ABB RobotStudio station: DeskDome.rspag

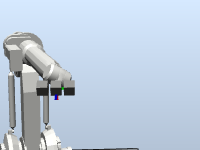
--- station ---
Station DeskDome (saved by RobotStudio 6.8.8148.134)
Controller DeskSystem
  mechanical unit ROB_1: IRB1410_5_144__01, 6 joints, base frame (0, 0, 0) mm
Layout (positions relative to the parent item):
  - IRB1410_5_144__01 [mechanism, from Robots\IRB1410_5_144_G_01.rslib] at (0, 0, 0) mm; joint values [0.3206, 0.0673, 0.0661, -0.5505, 0.5489, 0.6469] (rad or m)
  - 气缸3 [part] at (956.26, 325.16, 1145.27) mm, rotated rx -180 ry 60 rz 180 deg
  - 气缸2 [part] at (956.32, 263.96, 1145.39) mm, rotated rx -180 ry 60 rz 180 deg
  - 气缸1 [part] at (956.53, 200.68, 1145.75) mm, rotated rx -180 ry 60 rz 180 deg
  - 气缸运动 [smart component]
      signals: DI di_1, DI di_2, DI di_3, DO do_1, DO do_2, DO do_3, DI di_reset, DI di_M1, DI di_M2, DI di_M3, DO do_M1, DO do_M2, DO do_M3
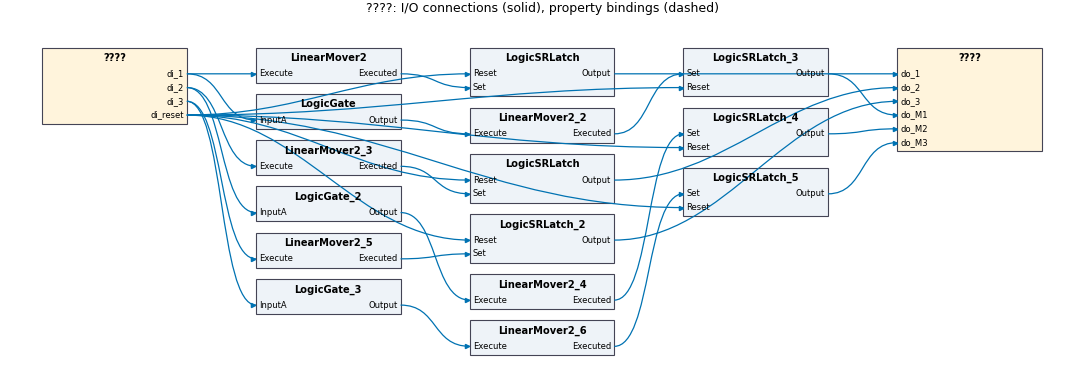
      connections:
        气缸运动.di_1 -> LinearMover2.Execute
        气缸运动.di_2 -> LinearMover2_3.Execute
        气缸运动.di_3 -> LinearMover2_5.Execute
        LogicSRLatch.Output -> 气缸运动.do_1
        气缸运动.di_reset -> LogicSRLatch.Reset
        LogicSRLatch.Output -> 气缸运动.do_2
        LogicSRLatch_2.Output -> 气缸运动.do_3
        气缸运动.di_reset -> LogicSRLatch.Reset
        气缸运动.di_reset -> LogicSRLatch_2.Reset
        LinearMover2.Executed -> LogicSRLatch.Set
        LinearMover2_2.Executed -> LogicSRLatch_3.Set
        气缸运动.di_reset -> LogicSRLatch_3.Reset
        LogicSRLatch_3.Output -> 气缸运动.do_M1
        LinearMover2_3.Executed -> LogicSRLatch.Set
        LinearMover2_4.Executed -> LogicSRLatch_4.Set
        气缸运动.di_reset -> LogicSRLatch_4.Reset
        LogicSRLatch_4.Output -> 气缸运动.do_M2
        LinearMover2_5.Executed -> LogicSRLatch_2.Set
        LinearMover2_6.Executed -> LogicSRLatch_5.Set
        气缸运动.di_reset -> LogicSRLatch_5.Reset
        LogicSRLatch_5.Output -> 气缸运动.do_M3
        气缸运动.di_1 -> LogicGate.InputA
        LogicGate.Output -> LinearMover2_2.Execute
        气缸运动.di_2 -> LogicGate_2.InputA
        LogicGate_2.Output -> LinearMover2_4.Execute
        气缸运动.di_3 -> LogicGate_3.InputA
        LogicGate_3.Output -> LinearMover2_6.Execute
    - LinearMover2 [smart component, from Components\LinearMover2.rslib]
        properties: Object=气缸1; Direction=[0 0 -0.01]; Distance=0.02; Duration=1; Reference=Global; ReferenceObject=(none)
    - LinearMover2_2 [smart component, from Components\LinearMover2.rslib]
        properties: Object=气缸1; Direction=[0 0 0.01]; Distance=0.02; Duration=1; Reference=Global; ReferenceObject=(none)
    - LinearMover2_3 [smart component, from Components\LinearMover2.rslib]
        properties: Object=气缸2; Direction=[0 0 -0.01]; Distance=0.02; Duration=1; Reference=Global; ReferenceObject=(none)
    - LinearMover2_4 [smart component, from Components\LinearMover2.rslib]
        properties: Object=气缸2; Direction=[0 0 0.01]; Distance=0.02; Duration=1; Reference=Global; ReferenceObject=(none)
    - LinearMover2_5 [smart component, from Components\LinearMover2.rslib]
        properties: Object=气缸3; Direction=[0 0 -0.01]; Distance=0.02; Duration=1; Reference=Global; ReferenceObject=(none)
    - LinearMover2_6 [smart component, from Components\LinearMover2.rslib]
        properties: Object=气缸3; Direction=[0 0 0.01]; Distance=0.02; Duration=1; Reference=Global; ReferenceObject=(none)
    - LogicSRLatch [smart component, from Components\LogicSRLatch.rslib]
    - LogicSRLatch [smart component, from Components\LogicSRLatch.rslib]
    - LogicSRLatch_2 [smart component, from Components\LogicSRLatch.rslib]
    - LogicSRLatch_3 [smart component, from Components\LogicSRLatch.rslib]
    - LogicSRLatch_4 [smart component, from Components\LogicSRLatch.rslib]
    - LogicSRLatch_5 [smart component, from Components\LogicSRLatch.rslib]
    - LogicGate [smart component, from Components\LogicGate.rslib]
        properties: Operator=NOT; Delay=0
    - LogicGate_2 [smart component, from Components\LogicGate.rslib]
        properties: Operator=NOT; Delay=0
    - LogicGate_3 [smart component, from Components\LogicGate.rslib]
        properties: Operator=NOT; Delay=0
Attachment: 气缸3 is attached to IRB1410_5_144__01 / Link6
Attachment: 气缸2 is attached to IRB1410_5_144__01 / Link6
Attachment: 气缸1 is attached to IRB1410_5_144__01 / Link6
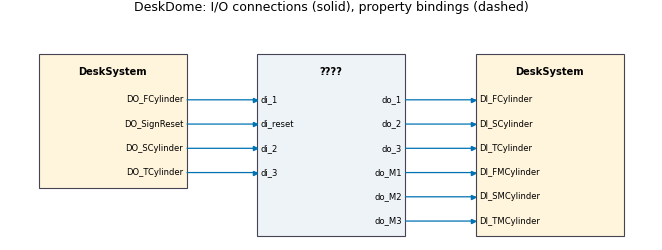
Station logic (signal -> signal, property => property):
  DeskSystem.DO_FCylinder -> 气缸运动.di_1
  气缸运动.do_1 -> DeskSystem.DI_FCylinder
  气缸运动.do_2 -> DeskSystem.DI_SCylinder
  气缸运动.do_3 -> DeskSystem.DI_TCylinder
  DeskSystem.DO_SignReset -> 气缸运动.di_reset
  DeskSystem.DO_SCylinder -> 气缸运动.di_2
  DeskSystem.DO_TCylinder -> 气缸运动.di_3
  气缸运动.do_M1 -> DeskSystem.DI_FMCylinder
  气缸运动.do_M2 -> DeskSystem.DI_SMCylinder
  气缸运动.do_M3 -> DeskSystem.DI_TMCylinder

--- Backups/DeskSystem/RAPID/TASK1/PROGMOD/Module1.mod ---
MODULE Module1

    !***********************************************************
    !
    ! Module:  Module1
    !
    ! Description:
    !   The seat test program is run with PC Sdk
    !
    ! Author: hanli
    !
    ! Version: 1.0
    !
    !***********************************************************


    !***********************************************************
    !
    ! Procedure main
    !
    !   This is the entry point of your program
    !
    !***********************************************************
    PROC main()
        TestNum:=0;
        InitializeSign;
        WHILE TestNum<MaxTestTimes DO
            DataIndex:=1;
            FOR Times FROM 1 TO 100 DO
                MoveRout DataIndex;
                IF MovePermis{DataIndex} THEN
                    TPWrite ""\Num:=DataIndex;
                ENDIF
                DataIndex:=DataIndex+1;
            ENDFOR
            TestNum:=TestNum+1;
        ENDWHILE
    ENDPROC

    PROC InitializeSign()
        Reset DO_FCylinder;
        Reset DO_SCylinder;
        Reset DO_TCylinder;
    ENDPROC

    PROC MoveRout(num rDataIndex)
        IF MovePermis{rDataIndex} THEN
            JudgeSignal DataIndex;
            MoveSpeed{DataIndex}.v_tcp:=NMoveSpeed{rDataIndex};
            MoveZone{rDataIndex}:=FZone(Zone);
            TEST MoveType{rDataIndex}
            CASE "MoveL":
                MoveL Point{rDataIndex},MoveSpeed{DataIndex},MoveZone{rDataIndex},tool0\WObj:=wobj0;
            CASE "MoveJ":
                MoveJ Point{rDataIndex},MoveSpeed{DataIndex},MoveZone{rDataIndex},tool0\WObj:=wobj0;
            CASE "MoveC":
                MoveC Point{rDataIndex},PointC{rDataIndex},MoveSpeed{DataIndex},MoveZone{rDataIndex},tool0\WObj:=wobj0;
            DEFAULT:
                MoveL Point{rDataIndex},MoveSpeed{DataIndex},MoveZone{rDataIndex},tool0\WObj:=wobj0;
            ENDTEST
            IF PressPermis{rDataIndex} THEN
                IF FirstPress THEN
                    FirstPoint:=CRobT();
                    MOffsetNum:=0;
                    WHILE SetForce{rDataIndex}<abs(Force_out_x) DO
                        MOffsetNum:=MOffsetNum+0.1;
                        MoveL RelTool(FirstPoint,0,0,MOffsetNum),v5,fine,tool0;
                    ENDWHILE
                    WHILE SetForce{rDataIndex}>abs(Force_out_x) DO
                        MOffsetNum:=MOffsetNum-0.1;
                        MoveL RelTool(FirstPoint,0,0,MOffsetNum),v5,fine,tool0;
                    ENDWHILE
                    Point{rDataIndex}:=CRobT();
                ENDIF
                Point{rDataIndex}.trans.x:=Point{rDataIndex}.trans.x+offestData(SetForce,rDataIndex);
            ENDIF
            Select_Action rDataIndex;
        ENDIF
    ENDPROC

    PROC Select_Action(INOUT num sDataIndex)
        IF SelectAction{sDataIndex,1} AND SelectAction{sDataIndex,2} AND SelectAction{sDataIndex,3} THEN
            Set DO_FCylinder;
            Set DO_SCylinder;
            Set DO_TCylinder;
            AllCJudge sDataIndex;
        ELSEIF SelectAction{sDataIndex,1} AND SelectAction{sDataIndex,2} THEN
            Set DO_FCylinder;
            Set DO_SCylinder;
            AllCJudge sDataIndex;
        ELSEIF SelectAction{sDataIndex,1} AND SelectAction{sDataIndex,3} THEN
            Set DO_FCylinder;
            Set DO_TCylinder;
            AllCJudge sDataIndex;
        ELSEIF SelectAction{sDataIndex,2} AND SelectAction{sDataIndex,3} THEN
            Set DO_SCylinder;
            Set DO_TCylinder;
            AllCJudge sDataIndex;
        ELSEIF SelectAction{sDataIndex,1} THEN
            Set DO_FCylinder;
            AllCJudge sDataIndex;
        ELSEIF SelectAction{sDataIndex,2} THEN
            Set DO_SCylinder;
            AllCJudge sDataIndex;
        ELSEIF SelectAction{sDataIndex,3} THEN
            Set DO_TCylinder;
            AllCJudge sDataIndex;
        ELSE
            AllCJudge sDataIndex;
        ENDIF

    ENDPROC

    FUNC num offestData(INOUT num oSetForce{*},INOUT num oDataIndex)
        offestNum:=0;
        IF oSetForce{oDataIndex}>abs(Force_out_x)+10 THEN
            offestNum:=offestNumData;
            FCDisBig:=true;
            IF oSetForce{oDataIndex}>abs(Force_out_x)+10 THEN
                offestNum:=0.1;
            ENDIF
        ELSEIF oSetForce{oDataIndex}<abs(Force_out_x)-10 THEN
            offestNum:=-offestNumData;
            FCDisSmall:=true;
            IF oSetForce{oDataIndex}<abs(Force_out_x)-10 THEN
                offestNum:=-0.1;
            ENDIF
        ENDIF
        PutOffestNum{oDataIndex}:=PutOffestNum{oDataIndex}+offestNum;
        IF PutOffestNum{oDataIndex}>=offestNumT OR PutOffestNum{oDataIndex}<=-offestNumT THEN
            Set OffestAlarmOn;
            Stop;
        ENDIF
        RETURN PutOffestNum{oDataIndex};
    ENDFUNC

    FUNC zonedata FZone(INOUT string FIndex{*})
        TEST FIndex{DataIndex}
        CASE "fine":
            RETURN fine;
        CASE "Z0":
            RETURN Z0;
        CASE "Z5":
            RETURN Z5;
        CASE "Z10":
            RETURN Z10;
        CASE "Z20":
            RETURN Z20;
        CASE "Z50":
            RETURN Z50;
        CASE "Z100":
            RETURN Z100;
        DEFAULT:
            RETURN Z1;
        ENDTEST
    ENDFUNC


    PROC AllCJudge(INOUT num sDataIndex)
        JudgeSign sDataIndex;
        Set DO_SignReset;
        JudgeSignReset sDataIndex;
        Reset DO_SignReset;
        Set DO_SignReset;
        JudgeMidSign sDataIndex;
        Reset DO_SignReset;
    ENDPROC

    PROC JudgeSign(INOUT num JDataIndex)
        IF JudgeWaitStartSign{JDataIndex,1}=FALSE THEN
            WaitDI DI_FCylinder,1;
        ENDIF
        IF JudgeWaitStartSign{JDataIndex,2}=FALSE THEN
            WaitDI DI_SCylinder,1;
        ENDIF
        IF JudgeWaitStartSign{JDataIndex,3}=FALSE THEN
            WaitDI DI_TCylinder,1;
        ENDIF
    ENDPROC

    PROC JudgeMidSign(INOUT num JDataIndex)
        IF JudgeWaitMidSign{JDataIndex,1}=FALSE THEN
            WaitDI DI_FMCylinder,1;
        ENDIF
        IF JudgeWaitMidSign{JDataIndex,2}=FALSE THEN
            WaitDI DI_SMCylinder,1;
        ENDIF
        IF JudgeWaitMidSign{JDataIndex,3}=FALSE THEN
            WaitDI DI_TMCylinder,1;
        ENDIF
    ENDPROC

    PROC JudgeSignReset(INOUT num JDataIndex)
        IF SelectActionReset{JDataIndex,1}=FALSE AND DO_FCylinder=1 THEN
            Reset DO_FCylinder;
        ENDIF
        IF SelectActionReset{JDataIndex,2}=FALSE AND DO_SCylinder=1 THEN
            Reset DO_SCylinder;
        ENDIF
        IF SelectActionReset{JDataIndex,3}=FALSE AND DO_TCylinder=1 THEN
            Reset DO_TCylinder;
        ENDIF
    ENDPROC

    PROC JudgeSignal(Inout num JDataIndex)
        VAR string WaitSignal;
        IF StrLen(JudgeWaitSignal{JDataIndex})>0 THEN
            i:=1;
            WaitSignal:="";
            FOR Judge FROM 1 TO StrLen(JudgeWaitSignal{JDataIndex}) DO
                WaitSignal:=StrPart(JudgeWaitSignal{JDataIndex},I,1);
                TEST WaitSignal
                CASE "1":
                    WaitDI DI_CarReady,1;
                CASE "2":
                    WaitDI DI_CarWindowOpen,1;
                CASE "3":
                    WaitDI DI_PLCOK,1;
                DEFAULT:
                ENDTEST
                i:=i+1;
            ENDFOR

        ENDIF


    ENDPROC


ENDMODULE

--- Backups/DeskSystem/RAPID/TASK1/PROGMOD/Module2.mod ---
MODULE Module2
	PROC Routine1()
		DataIndex := 1;
		FOR qq FROM 1 TO 99 DO
            JudgeSignal DataIndex;
			DataIndex := DataIndex + 1;
		ENDFOR
		TPWrite ""\Num:=DataIndex;
	ENDPROC

    PROC textR()
        WaitTime 100000;
    ENDPROC

ENDMODULE

--- Backups/DeskSystem/RAPID/TASK1/PROGMOD/RobotData.mod ---
MODULE RobotData
    !========================Array content=========================================
    PERS robtarget Point{100}:=[[[943.61,0,1152.5],[0.5,6.23716E-9,0.866025,3.60103E-9],[0,0,0,0],[9E+9,9E+9,9E+9,9E+9,9E+9,9E+9]],[[943.61,-325.96,1152.5],[0.5,2.44722E-8,0.866025,4.68183E-8],[-1,0,-1,0],[9E+9,9E+9,9E+9,9E+9,9E+9,9E+9]],[[943.61,209.03,1152.5],[0.5,3.78656E-8,0.866025,-2.06236E-8],[0,-1,0,0],[9E+9,9E+9,9E+9,9E+9,9E+9,9E+9]],[[943.61,209.03,857.09],[0.5,9.49976E-8,0.866025,6.72883E-8],[0,-1,0,0],[9E+9,9E+9,9E+9,9E+9,9E+9,9E+9]],[[943.61,-465.67,857.09],[0.5,-4.15323E-9,0.866025,6.47384E-8],[-1,0,-1,0],[9E+9,9E+9,9E+9,9E+9,9E+9,9E+9]],[[943.61,734.61,857.09],[0.5,4.60295E-8,0.866025,2.22463E-8],[0,-1,0,0],[9E+9,9E+9,9E+9,9E+9,9E+9,9E+9]],[[943.61,734.61,1027.54],[0.5,4.43579E-8,0.866025,1.33957E-9],[0,-1,0,0],[9E+9,9E+9,9E+9,9E+9,9E+9,9E+9]],[[943.61,0,1152.5],[0.5,6.23717E-9,0.866025,3.60103E-9],[0,0,0,0],[9E+9,9E+9,9E+9,9E+9,9E+9,9E+9]],[[943.61,0,1152.5],[0.5,6.23717E-9,0.866025,3.60103E-9],[0,0,0,0],[9E+9,9E+9,9E+9,9E+9,9E+9,9E+9]],[[943.61,0,1152.5],[0.5,6.23717E-9,0.866025,3.60103E-9],[0,0,0,0],[9E+9,9E+9,9E+9,9E+9,9E+9,9E+9]],[[943.61,0,1152.5],[0.5,6.23717E-9,0.866025,3.60103E-9],[0,0,0,0],[9E+9,9E+9,9E+9,9E+9,9E+9,9E+9]],[[943.61,0,1152.5],[0.5,6.23717E-9,0.866025,3.60103E-9],[0,0,0,0],[9E+9,9E+9,9E+9,9E+9,9E+9,9E+9]],[[943.61,0,1152.5],[0.5,6.23717E-9,0.866025,3.60103E-9],[0,0,0,0],[9E+9,9E+9,9E+9,9E+9,9E+9,9E+9]],[[943.61,0,1152.5],[0.5,6.23717E-9,0.866025,3.60103E-9],[0,0,0,0],[9E+9,9E+9,9E+9,9E+9,9E+9,9E+9]],[[943.61,0,1152.5],[0.5,6.23717E-9,0.866025,3.60103E-9],[0,0,0,0],[9E+9,9E+9,9E+9,9E+9,9E+9,9E+9]],[[943.61,0,1152.5],[0.5,6.23717E-9,0.866025,3.60103E-9],[0,0,0,0],[9E+9,9E+9,9E+9,9E+9,9E+9,9E+9]],[[943.61,0,1152.5],[0.5,6.23717E-9,0.866025,3.60103E-9],[0,0,0,0],[9E+9,9E+9,9E+9,9E+9,9E+9,9E+9]],[[943.61,0,1152.5],[0.5,6.23717E-9,0.866025,3.60103E-9],[0,0,0,0],[9E+9,9E+9,9E+9,9E+9,9E+9,9E+9]],[[943.61,0,1152.5],[0.5,6.23717E-9,0.866025,3.60103E-9],[0,0,0,0],[9E+9,9E+9,9E+9,9E+9,9E+9,9E+9]],[[943.61,0,1152.5],[0.5,6.23717E-9,0.866025,3.60103E-9],[0,0,0,0],[9E+9,9E+9,9E+9,9E+9,9E+9,9E+9]],[[943.61,0,1152.5],[0.5,6.23717E-9,0.866025,3.60103E-9],[0,0,0,0],[9E+9,9E+9,9E+9,9E+9,9E+9,9E+9]],[[943.61,0,1152.5],[0.5,6.23717E-9,0.866025,3.60103E-9],[0,0,0,0],[9E+9,9E+9,9E+9,9E+9,9E+9,9E+9]],[[943.61,0,1152.5],[0.5,6.23717E-9,0.866025,3.60103E-9],[0,0,0,0],[9E+9,9E+9,9E+9,9E+9,9E+9,9E+9]],[[943.61,0,1152.5],[0.5,6.23717E-9,0.866025,3.60103E-9],[0,0,0,0],[9E+9,9E+9,9E+9,9E+9,9E+9,9E+9]],[[943.61,0,1152.5],[0.5,6.23717E-9,0.866025,3.60103E-9],[0,0,0,0],[9E+9,9E+9,9E+9,9E+9,9E+9,9E+9]],[[943.61,0,1152.5],[0.5,6.23717E-9,0.866025,3.60103E-9],[0,0,0,0],[9E+9,9E+9,9E+9,9E+9,9E+9,9E+9]],[[943.61,0,1152.5],[0.5,6.23717E-9,0.866025,3.60103E-9],[0,0,0,0],[9E+9,9E+9,9E+9,9E+9,9E+9,9E+9]],[[943.61,0,1152.5],[0.5,6.23717E-9,0.866025,3.60103E-9],[0,0,0,0],[9E+9,9E+9,9E+9,9E+9,9E+9,9E+9]],[[943.61,0,1152.5],[0.5,6.23717E-9,0.866025,3.60103E-9],[0,0,0,0],[9E+9,9E+9,9E+9,9E+9,9E+9,9E+9]],[[943.61,0,1152.5],[0.5,6.23717E-9,0.866025,3.60103E-9],[0,0,0,0],[9E+9,9E+9,9E+9,9E+9,9E+9,9E+9]],[[943.61,0,1152.5],[0.5,6.23717E-9,0.866025,3.60103E-9],[0,0,0,0],[9E+9,9E+9,9E+9,9E+9,9E+9,9E+9]],[[943.61,0,1152.5],[0.5,6.23717E-9,0.866025,3.60103E-9],[0,0,0,0],[9E+9,9E+9,9E+9,9E+9,9E+9,9E+9]],[[943.61,0,1152.5],[0.5,6.23717E-9,0.866025,3.60103E-9],[0,0,0,0],[9E+9,9E+9,9E+9,9E+9,9E+9,9E+9]],[[943.61,0,1152.5],[0.5,6.23717E-9,0.866025,3.60103E-9],[0,0,0,0],[9E+9,9E+9,9E+9,9E+9,9E+9,9E+9]],[[943.61,0,1152.5],[0.5,6.23717E-9,0.866025,3.60103E-9],[0,0,0,0],[9E+9,9E+9,9E+9,9E+9,9E+9,9E+9]],[[943.61,0,1152.5],[0.5,6.23717E-9,0.866025,3.60103E-9],[0,0,0,0],[9E+9,9E+9,9E+9,9E+9,9E+9,9E+9]],[[943.61,0,1152.5],[0.5,6.23717E-9,0.866025,3.60103E-9],[0,0,0,0],[9E+9,9E+9,9E+9,9E+9,9E+9,9E+9]],[[943.61,0,1152.5],[0.5,6.23717E-9,0.866025,3.60103E-9],[0,0,0,0],[9E+9,9E+9,9E+9,9E+9,9E+9,9E+9]],[[943.61,0,1152.5],[0.5,6.23717E-9,0.866025,3.60103E-9],[0,0,0,0],[9E+9,9E+9,9E+9,9E+9,9E+9,9E+9]],[[943.61,0,1152.5],[0.5,6.23717E-9,0.866025,3.60103E-9],[0,0,0,0],[9E+9,9E+9,9E+9,9E+9,9E+9,9E+9]],[[943.61,0,1152.5],[0.5,6.23717E-9,0.866025,3.60103E-9],[0,0,0,0],[9E+9,9E+9,9E+9,9E+9,9E+9,9E+9]],[[943.61,0,1152.5],[0.5,6.23717E-9,0.866025,3.60103E-9],[0,0,0,0],[9E+9,9E+9,9E+9,9E+9,9E+9,9E+9]],[[943.61,0,1152.5],[0.5,6.23717E-9,0.866025,3.60103E-9],[0,0,0,0],[9E+9,9E+9,9E+9,9E+9,9E+9,9E+9]],[[943.61,0,1152.5],[0.5,6.23717E-9,0.866025,3.60103E-9],[0,0,0,0],[9E+9,9E+9,9E+9,9E+9,9E+9,9E+9]],[[943.61,0,1152.5],[0.5,6.23717E-9,0.866025,3.60103E-9],[0,0,0,0],[9E+9,9E+9,9E+9,9E+9,9E+9,9E+9]],[[943.61,0,1152.5],[0.5,6.23717E-9,0.866025,3.60103E-9],[0,0,0,0],[9E+9,9E+9,9E+9,9E+9,9E+9,9E+9]],[[943.61,0,1152.5],[0.5,6.23717E-9,0.866025,3.60103E-9],[0,0,0,0],[9E+9,9E+9,9E+9,9E+9,9E+9,9E+9]],[[943.61,0,1152.5],[0.5,6.23717E-9,0.866025,3.60103E-9],[0,0,0,0],[9E+9,9E+9,9E+9,9E+9,9E+9,9E+9]],[[943.61,0,1152.5],[0.5,6.23717E-9,0.866025,3.60103E-9],[0,0,0,0],[9E+9,9E+9,9E+9,9E+9,9E+9,9E+9]],[[943.61,0,1152.5],[0.5,6.23717E-9,0.866025,3.60103E-9],[0,0,0,0],[9E+9,9E+9,9E+9,9E+9,9E+9,9E+9]],[[943.61,0,1152.5],[0.5,6.23717E-9,0.866025,3.60103E-9],[0,0,0,0],[9E+9,9E+9,9E+9,9E+9,9E+9,9E+9]],[[943.61,0,1152.5],[0.5,6.23717E-9,0.866025,3.60103E-9],[0,0,0,0],[9E+9,9E+9,9E+9,9E+9,9E+9,9E+9]],[[943.61,0,1152.5],[0.5,6.23717E-9,0.866025,3.60103E-9],[0,0,0,0],[9E+9,9E+9,9E+9,9E+9,9E+9,9E+9]],[[943.61,0,1152.5],[0.5,6.23717E-9,0.866025,3.60103E-9],[0,0,0,0],[9E+9,9E+9,9E+9,9E+9,9E+9,9E+9]],[[943.61,0,1152.5],[0.5,6.23717E-9,0.866025,3.60103E-9],[0,0,0,0],[9E+9,9E+9,9E+9,9E+9,9E+9,9E+9]],[[943.61,0,1152.5],[0.5,6.23717E-9,0.866025,3.60103E-9],[0,0,0,0],[9E+9,9E+9,9E+9,9E+9,9E+9,9E+9]],[[943.61,0,1152.5],[0.5,6.23717E-9,0.866025,3.60103E-9],[0,0,0,0],[9E+9,9E+9,9E+9,9E+9,9E+9,9E+9]],[[943.61,0,1152.5],[0.5,6.23717E-9,0.866025,3.60103E-9],[0,0,0,0],[9E+9,9E+9,9E+9,9E+9,9E+9,9E+9]],[[943.61,0,1152.5],[0.5,6.23717E-9,0.866025,3.60103E-9],[0,0,0,0],[9E+9,9E+9,9E+9,9E+9,9E+9,9E+9]],[[943.61,0,1152.5],[0.5,6.23717E-9,0.866025,3.60103E-9],[0,0,0,0],[9E+9,9E+9,9E+9,9E+9,9E+9,9E+9]],[[943.61,0,1152.5],[0.5,6.23717E-9,0.866025,3.60103E-9],[0,0,0,0],[9E+9,9E+9,9E+9,9E+9,9E+9,9E+9]],[[943.61,0,1152.5],[0.5,6.23717E-9,0.866025,3.60103E-9],[0,0,0,0],[9E+9,9E+9,9E+9,9E+9,9E+9,9E+9]],[[943.61,0,1152.5],[0.5,6.23717E-9,0.866025,3.60103E-9],[0,0,0,0],[9E+9,9E+9,9E+9,9E+9,9E+9,9E+9]],[[943.61,0,1152.5],[0.5,6.23717E-9,0.866025,3.60103E-9],[0,0,0,0],[9E+9,9E+9,9E+9,9E+9,9E+9,9E+9]],[[943.61,0,1152.5],[0.5,6.23717E-9,0.866025,3.60103E-9],[0,0,0,0],[9E+9,9E+9,9E+9,9E+9,9E+9,9E+9]],[[943.61,0,1152.5],[0.5,6.23717E-9,0.866025,3.60103E-9],[0,0,0,0],[9E+9,9E+9,9E+9,9E+9,9E+9,9E+9]],[[943.61,0,1152.5],[0.5,6.23717E-9,0.866025,3.60103E-9],[0,0,0,0],[9E+9,9E+9,9E+9,9E+9,9E+9,9E+9]],[[943.61,0,1152.5],[0.5,6.23717E-9,0.866025,3.60103E-9],[0,0,0,0],[9E+9,9E+9,9E+9,9E+9,9E+9,9E+9]],[[943.61,0,1152.5],[0.5,6.23717E-9,0.866025,3.60103E-9],[0,0,0,0],[9E+9,9E+9,9E+9,9E+9,9E+9,9E+9]],[[943.61,0,1152.5],[0.5,6.23717E-9,0.866025,3.60103E-9],[0,0,0,0],[9E+9,9E+9,9E+9,9E+9,9E+9,9E+9]],[[943.61,0,1152.5],[0.5,6.23717E-9,0.866025,3.60103E-9],[0,0,0,0],[9E+9,9E+9,9E+9,9E+9,9E+9,9E+9]],[[943.61,0,1152.5],[0.5,6.23717E-9,0.866025,3.60103E-9],[0,0,0,0],[9E+9,9E+9,9E+9,9E+9,9E+9,9E+9]],[[943.61,0,1152.5],[0.5,6.23717E-9,0.866025,3.60103E-9],[0,0,0,0],[9E+9,9E+9,9E+9,9E+9,9E+9,9E+9]],[[943.61,0,1152.5],[0.5,6.23717E-9,0.866025,3.60103E-9],[0,0,0,0],[9E+9,9E+9,9E+9,9E+9,9E+9,9E+9]],[[943.61,0,1152.5],[0.5,6.23717E-9,0.866025,3.60103E-9],[0,0,0,0],[9E+9,9E+9,9E+9,9E+9,9E+9,9E+9]],[[943.61,0,1152.5],[0.5,6.23717E-9,0.866025,3.60103E-9],[0,0,0,0],[9E+9,9E+9,9E+9,9E+9,9E+9,9E+9]],[[943.61,0,1152.5],[0.5,6.23717E-9,0.866025,3.60103E-9],[0,0,0,0],[9E+9,9E+9,9E+9,9E+9,9E+9,9E+9]],[[943.61,0,1152.5],[0.5,6.23717E-9,0.866025,3.60103E-9],[0,0,0,0],[9E+9,9E+9,9E+9,9E+9,9E+9,9E+9]],[[943.61,0,1152.5],[0.5,6.23717E-9,0.866025,3.60103E-9],[0,0,0,0],[9E+9,9E+9,9E+9,9E+9,9E+9,9E+9]],[[943.61,0,1152.5],[0.5,6.23717E-9,0.866025,3.60103E-9],[0,0,0,0],[9E+9,9E+9,9E+9,9E+9,9E+9,9E+9]],[[943.61,0,1152.5],[0.5,6.23717E-9,0.866025,3.60103E-9],[0,0,0,0],[9E+9,9E+9,9E+9,9E+9,9E+9,9E+9]],[[943.61,0,1152.5],[0.5,6.23717E-9,0.866025,3.60103E-9],[0,0,0,0],[9E+9,9E+9,9E+9,9E+9,9E+9,9E+9]],[[943.61,0,1152.5],[0.5,6.23717E-9,0.866025,3.60103E-9],[0,0,0,0],[9E+9,9E+9,9E+9,9E+9,9E+9,9E+9]],[[943.61,0,1152.5],[0.5,6.23717E-9,0.866025,3.60103E-9],[0,0,0,0],[9E+9,9E+9,9E+9,9E+9,9E+9,9E+9]],[[943.61,0,1152.5],[0.5,6.23717E-9,0.866025,3.60103E-9],[0,0,0,0],[9E+9,9E+9,9E+9,9E+9,9E+9,9E+9]],[[943.61,0,1152.5],[0.5,6.23717E-9,0.866025,3.60103E-9],[0,0,0,0],[9E+9,9E+9,9E+9,9E+9,9E+9,9E+9]],[[943.61,0,1152.5],[0.5,6.23717E-9,0.866025,3.60103E-9],[0,0,0,0],[9E+9,9E+9,9E+9,9E+9,9E+9,9E+9]],[[943.61,0,1152.5],[0.5,6.23717E-9,0.866025,3.60103E-9],[0,0,0,0],[9E+9,9E+9,9E+9,9E+9,9E+9,9E+9]],[[943.61,0,1152.5],[0.5,6.23717E-9,0.866025,3.60103E-9],[0,0,0,0],[9E+9,9E+9,9E+9,9E+9,9E+9,9E+9]],[[943.61,0,1152.5],[0.5,6.23717E-9,0.866025,3.60103E-9],[0,0,0,0],[9E+9,9E+9,9E+9,9E+9,9E+9,9E+9]],[[943.61,0,1152.5],[0.5,6.23717E-9,0.866025,3.60103E-9],[0,0,0,0],[9E+9,9E+9,9E+9,9E+9,9E+9,9E+9]],[[943.61,0,1152.5],[0.5,6.23717E-9,0.866025,3.60103E-9],[0,0,0,0],[9E+9,9E+9,9E+9,9E+9,9E+9,9E+9]],[[943.61,0,1152.5],[0.5,6.23717E-9,0.866025,3.60103E-9],[0,0,0,0],[9E+9,9E+9,9E+9,9E+9,9E+9,9E+9]],[[943.61,0,1152.5],[0.5,6.23717E-9,0.866025,3.60103E-9],[0,0,0,0],[9E+9,9E+9,9E+9,9E+9,9E+9,9E+9]],[[943.61,0,1152.5],[0.5,6.23717E-9,0.866025,3.60103E-9],[0,0,0,0],[9E+9,9E+9,9E+9,9E+9,9E+9,9E+9]],[[943.61,0,1152.5],[0.5,6.23717E-9,0.866025,3.60103E-9],[0,0,0,0],[9E+9,9E+9,9E+9,9E+9,9E+9,9E+9]],[[943.61,0,1152.5],[0.5,6.23717E-9,0.866025,3.60103E-9],[0,0,0,0],[9E+9,9E+9,9E+9,9E+9,9E+9,9E+9]],[[943.61,0,1152.5],[0.5,6.23717E-9,0.866025,3.60103E-9],[0,0,0,0],[9E+9,9E+9,9E+9,9E+9,9E+9,9E+9]],[[943.61,0,1152.5],[0.5,6.23717E-9,0.866025,3.60103E-9],[0,0,0,0],[9E+9,9E+9,9E+9,9E+9,9E+9,9E+9]],[[943.61,0,1152.5],[0.5,6.23717E-9,0.866025,3.60103E-9],[0,0,0,0],[9E+9,9E+9,9E+9,9E+9,9E+9,9E+9]]];
    PERS speeddata MoveSpeed{100}:=[[200,500,5000,1000],[50,500,5000,1000],[200,500,5000,1000],[200,500,5000,1000],[400,500,5000,1000],[400,500,5000,1000],[400,500,5000,1000],[200,500,5000,1000],[50,500,5000,1000],[200,500,5000,1000],[200,500,5000,1000],[200,500,5000,1000],[200,500,5000,1000],[1000,500,5000,1000],[1000,500,5000,1000],[1000,500,5000,1000],[1000,500,5000,1000],[1000,500,5000,1000],[1000,500,5000,1000],[1000,500,5000,1000],[1000,500,5000,1000],[1000,500,5000,1000],[1000,500,5000,1000],[1000,500,5000,1000],[1000,500,5000,1000],[1000,500,5000,1000],[1000,500,5000,1000],[1000,500,5000,1000],[1000,500,5000,1000],[1000,500,5000,1000],[1000,500,5000,1000],[1000,500,5000,1000],[1000,500,5000,1000],[1000,500,5000,1000],[1000,500,5000,1000],[1000,500,5000,1000],[1000,500,5000,1000],[1000,500,5000,1000],[1000,500,5000,1000],[1000,500,5000,1000],[1000,500,5000,1000],[1000,500,5000,1000],[1000,500,5000,1000],[1000,500,5000,1000],[1000,500,5000,1000],[1000,500,5000,1000],[1000,500,5000,1000],[1000,500,5000,1000],[1000,500,5000,1000],[1000,500,5000,1000],[1000,500,5000,1000],[1000,500,5000,1000],[1000,500,5000,1000],[1000,500,5000,1000],[1000,500,5000,1000],[1000,500,5000,1000],[1000,500,5000,1000],[1000,500,5000,1000],[1000,500,5000,1000],[1000,500,5000,1000],[1000,500,5000,1000],[1000,500,5000,1000],[1000,500,5000,1000],[1000,500,5000,1000],[1000,500,5000,1000],[1000,500,5000,1000],[1000,500,5000,1000],[1000,500,5000,1000],[1000,500,5000,1000],[1000,500,5000,1000],[1000,500,5000,1000],[1000,500,5000,1000],[1000,500,5000,1000],[1000,500,5000,1000],[1000,500,5000,1000],[1000,500,5000,1000],[1000,500,5000,1000],[1000,500,5000,1000],[1000,500,5000,1000],[1000,500,5000,1000],[1000,500,5000,1000],[1000,500,5000,1000],[1000,500,5000,1000],[1000,500,5000,1000],[1000,500,5000,1000],[1000,500,5000,1000],[1000,500,5000,1000],[1000,500,5000,1000],[1000,500,5000,1000],[1000,500,5000,1000],[1000,500,5000,1000],[1000,500,5000,1000],[1000,500,5000,1000],[1000,500,5000,1000],[1000,500,5000,1000],[1000,500,5000,1000],[1000,500,5000,1000],[1000,500,5000,1000],[1000,500,5000,1000],[1000,500,5000,1000]];
    PERS zonedata MoveZone{100}:=[[TRUE,0,0,0,0,0,0],[TRUE,0,0,0,0,0,0],[TRUE,0,0,0,0,0,0],[TRUE,0,0,0,0,0,0],[FALSE,0.3,0.3,0.3,0.03,0.3,0.03],[FALSE,50,75,75,7.5,75,7.5],[FALSE,100,150,150,15,150,15],[TRUE,0,0,0,0,0,0],[TRUE,0,0,0,0,0,0],[TRUE,0,0,0,0,0,0],[TRUE,0,0,0,0,0,0],[TRUE,0,0,0,0,0,0],[TRUE,0,0,0,0,0,0],[FALSE,50,75,75,7.5,75,7.5],[FALSE,50,75,75,7.5,75,7.5],[FALSE,50,75,75,7.5,75,7.5],[FALSE,50,75,75,7.5,75,7.5],[FALSE,50,75,75,7.5,75,7.5],[FALSE,50,75,75,7.5,75,7.5],[FALSE,50,75,75,7.5,75,7.5],[FALSE,50,75,75,7.5,75,7.5],[FALSE,50,75,75,7.5,75,7.5],[FALSE,50,75,75,7.5,75,7.5],[FALSE,50,75,75,7.5,75,7.5],[FALSE,50,75,75,7.5,75,7.5],[FALSE,50,75,75,7.5,75,7.5],[FALSE,50,75,75,7.5,75,7.5],[FALSE,50,75,75,7.5,75,7.5],[FALSE,50,75,75,7.5,75,7.5],[FALSE,50,75,75,7.5,75,7.5],[FALSE,50,75,75,7.5,75,7.5],[FALSE,50,75,75,7.5,75,7.5],[FALSE,50,75,75,7.5,75,7.5],[FALSE,50,75,75,7.5,75,7.5],[FALSE,50,75,75,7.5,75,7.5],[FALSE,50,75,75,7.5,75,7.5],[FALSE,50,75,75,7.5,75,7.5],[FALSE,50,75,75,7.5,75,7.5],[FALSE,50,75,75,7.5,75,7.5],[FALSE,50,75,75,7.5,75,7.5],[FALSE,50,75,75,7.5,75,7.5],[FALSE,50,75,75,7.5,75,7.5],[FALSE,50,75,75,7.5,75,7.5],[FALSE,50,75,75,7.5,75,7.5],[FALSE,50,75,75,7.5,75,7.5],[FALSE,50,75,75,7.5,75,7.5],[FALSE,50,75,75,7.5,75,7.5],[FALSE,50,75,75,7.5,75,7.5],[FALSE,50,75,75,7.5,75,7.5],[FALSE,50,75,75,7.5,75,7.5],[FALSE,50,75,75,7.5,75,7.5],[FALSE,50,75,75,7.5,75,7.5],[FALSE,50,75,75,7.5,75,7.5],[FALSE,50,75,75,7.5,75,7.5],[FALSE,50,75,75,7.5,75,7.5],[FALSE,50,75,75,7.5,75,7.5],[FALSE,50,75,75,7.5,75,7.5],[FALSE,50,75,75,7.5,75,7.5],[FALSE,50,75,75,7.5,75,7.5],[FALSE,50,75,75,7.5,75,7.5],[FALSE,50,75,75,7.5,75,7.5],[FALSE,50,75,75,7.5,75,7.5],[FALSE,50,75,75,7.5,75,7.5],[FALSE,50,75,75,7.5,75,7.5],[FALSE,50,75,75,7.5,75,7.5],[FALSE,50,75,75,7.5,75,7.5],[FALSE,50,75,75,7.5,75,7.5],[FALSE,50,75,75,7.5,75,7.5],[FALSE,50,75,75,7.5,75,7.5],[FALSE,50,75,75,7.5,75,7.5],[FALSE,50,75,75,7.5,75,7.5],[FALSE,50,75,75,7.5,75,7.5],[FALSE,50,75,75,7.5,75,7.5],[FALSE,50,75,75,7.5,75,7.5],[FALSE,50,75,75,7.5,75,7.5],[FALSE,50,75,75,7.5,75,7.5],[FALSE,50,75,75,7.5,75,7.5],[FALSE,50,75,75,7.5,75,7.5],[FALSE,50,75,75,7.5,75,7.5],[FALSE,50,75,75,7.5,75,7.5],[FALSE,50,75,75,7.5,75,7.5],[FALSE,50,75,75,7.5,75,7.5],[FALSE,50,75,75,7.5,75,7.5],[FALSE,50,75,75,7.5,75,7.5],[FALSE,50,75,75,7.5,75,7.5],[FALSE,50,75,75,7.5,75,7.5],[FALSE,50,75,75,7.5,75,7.5],[FALSE,50,75,75,7.5,75,7.5],[FALSE,50,75,75,7.5,75,7.5],[FALSE,50,75,75,7.5,75,7.5],[FALSE,50,75,75,7.5,75,7.5],[FALSE,50,75,75,7.5,75,7.5],[FALSE,50,75,75,7.5,75,7.5],[FALSE,50,75,75,7.5,75,7.5],[FALSE,50,75,75,7.5,75,7.5],[FALSE,50,75,75,7.5,75,7.5],[FALSE,50,75,75,7.5,75,7.5],[FALSE,50,75,75,7.5,75,7.5],[FALSE,50,75,75,7.5,75,7.5],[FALSE,50,75,75,7.5,75,7.5]];
    PERS num SetForce{100}:=[100,100,100,100,100,100,100,100,100,100,100,100,100,0,0,0,0,0,0,0,0,0,0,0,0,0,0,0,0,0,0,0,0,0,0,0,0,0,0,0,0,0,0,0,0,0,0,0,0,0,0,0,0,0,0,0,0,0,0,0,0,0,0,0,0,0,0,0,0,0,0,0,0,0,0,0,0,0,0,0,0,0,0,0,0,0,0,0,0,0,0,0,0,0,0,0,0,0,0,0];
    PERS bool SelectAction{100,3}:=[[TRUE,TRUE,TRUE],[TRUE,FALSE,FALSE],[TRUE,TRUE,FALSE],[FALSE,TRUE,FALSE],[FALSE,FALSE,FALSE],[FALSE,FALSE,FALSE],[FALSE,FALSE,TRUE],[FALSE,FALSE,TRUE],[FALSE,FALSE,FALSE],[FALSE,FALSE,FALSE],[TRUE,FALSE,FALSE],[FALSE,FALSE,FALSE],[FALSE,FALSE,FALSE],[FALSE,FALSE,FALSE],[FALSE,FALSE,FALSE],[FALSE,FALSE,FALSE],[FALSE,FALSE,FALSE],[FALSE,FALSE,FALSE],[FALSE,FALSE,FALSE],[FALSE,FALSE,FALSE],[FALSE,FALSE,FALSE],[FALSE,FALSE,FALSE],[FALSE,FALSE,FALSE],[FALSE,FALSE,FALSE],[FALSE,FALSE,FALSE],[FALSE,FALSE,FALSE],[FALSE,FALSE,FALSE],[FALSE,FALSE,FALSE],[FALSE,FALSE,FALSE],[FALSE,FALSE,FALSE],[FALSE,FALSE,FALSE],[FALSE,FALSE,FALSE],[FALSE,FALSE,FALSE],[FALSE,FALSE,FALSE],[FALSE,FALSE,FALSE],[FALSE,FALSE,FALSE],[FALSE,FALSE,FALSE],[FALSE,FALSE,FALSE],[FALSE,FALSE,FALSE],[FALSE,FALSE,FALSE],[FALSE,FALSE,FALSE],[FALSE,FALSE,FALSE],[FALSE,FALSE,FALSE],[FALSE,FALSE,FALSE],[FALSE,FALSE,FALSE],[FALSE,FALSE,FALSE],[FALSE,FALSE,FALSE],[FALSE,FALSE,FALSE],[FALSE,FALSE,FALSE],[FALSE,FALSE,FALSE],[FALSE,FALSE,FALSE],[FALSE,FALSE,FALSE],[FALSE,FALSE,FALSE],[FALSE,FALSE,FALSE],[FALSE,FALSE,FALSE],[FALSE,FALSE,FALSE],[FALSE,FALSE,FALSE],[FALSE,FALSE,FALSE],[FALSE,FALSE,FALSE],[FALSE,FALSE,FALSE],[FALSE,FALSE,FALSE],[FALSE,FALSE,FALSE],[FALSE,FALSE,FALSE],[FALSE,FALSE,FALSE],[FALSE,FALSE,FALSE],[FALSE,FALSE,FALSE],[FALSE,FALSE,FALSE],[FALSE,FALSE,FALSE],[FALSE,FALSE,FALSE],[FALSE,FALSE,FALSE],[FALSE,FALSE,FALSE],[FALSE,FALSE,FALSE],[FALSE,FALSE,FALSE],[FALSE,FALSE,FALSE],[FALSE,FALSE,FALSE],[FALSE,FALSE,FALSE],[FALSE,FALSE,FALSE],[FALSE,FALSE,FALSE],[FALSE,FALSE,FALSE],[FALSE,FALSE,FALSE],[FALSE,FALSE,FALSE],[FALSE,FALSE,FALSE],[FALSE,FALSE,FALSE],[FALSE,FALSE,FALSE],[FALSE,FALSE,FALSE],[FALSE,FALSE,FALSE],[FALSE,FALSE,FALSE],[FALSE,FALSE,FALSE],[FALSE,FALSE,FALSE],[FALSE,FALSE,FALSE],[FALSE,FALSE,FALSE],[FALSE,FALSE,FALSE],[FALSE,FALSE,FALSE],[FALSE,FALSE,FALSE],[FALSE,FALSE,FALSE],[FALSE,FALSE,FALSE],[FALSE,FALSE,FALSE],[FALSE,FALSE,FALSE],[FALSE,FALSE,FALSE],[FALSE,FALSE,FALSE]];
    PERS bool MovePermis{100}:=[TRUE,TRUE,TRUE,TRUE,TRUE,TRUE,TRUE,TRUE,TRUE,TRUE,TRUE,TRUE,TRUE,FALSE,FALSE,FALSE,FALSE,FALSE,FALSE,FALSE,FALSE,FALSE,FALSE,FALSE,FALSE,FALSE,FALSE,FALSE,FALSE,FALSE,FALSE,FALSE,FALSE,FALSE,FALSE,FALSE,FALSE,FALSE,FALSE,FALSE,FALSE,FALSE,FALSE,FALSE,FALSE,FALSE,FALSE,FALSE,FALSE,FALSE,FALSE,FALSE,FALSE,FALSE,FALSE,FALSE,FALSE,FALSE,FALSE,FALSE,FALSE,FALSE,FALSE,FALSE,FALSE,FALSE,FALSE,FALSE,FALSE,FALSE,FALSE,FALSE,FALSE,FALSE,FALSE,FALSE,FALSE,FALSE,FALSE,FALSE,FALSE,FALSE,FALSE,FALSE,FALSE,FALSE,FALSE,FALSE,FALSE,FALSE,FALSE,FALSE,FALSE,FALSE,FALSE,FALSE,FALSE,FALSE,FALSE,FALSE];
    PERS num NMoveSpeed{100}:=[20,50,60,200,600,300,400,200,50,200,200,200,200,0,0,0,0,0,0,0,0,0,0,0,0,0,0,0,0,0,0,0,0,0,0,0,0,0,0,0,0,0,0,0,0,0,0,0,0,0,0,0,0,0,0,0,0,0,0,0,0,0,0,0,0,0,0,0,0,0,0,0,0,0,0,0,0,0,0,0,0,0,0,0,0,0,0,0,0,0,0,0,0,0,0,0,0,0,0,0];
    PERS num NMoveZone{100}:=[0,0,0,0,0,0,0,0,0,0,0,0,0,0,0,0,0,0,0,0,0,0,0,0,0,0,0,0,0,0,0,0,0,0,0,0,0,0,0,0,0,0,0,0,0,0,0,0,0,0,0,0,0,0,0,0,0,0,0,0,0,0,0,0,0,0,0,0,0,0,0,0,0,0,0,0,0,0,0,0,0,0,0,0,0,0,0,0,0,0,0,0,0,0,0,0,0,0,0,0];
    PERS string Zone{100}:=["fine","fine","fine","fine","fine","fine","Z100","fine","fine","fine","fine","fine","fine","","","","","","","","","","","","","","","","","","","","","","","","","","","","","","","","","","","","","","","","","","","","","","","","","","","","","","","","","","","","","","","","","","","","","","","","","","","","","","","","","","","","","","",""];
    PERS bool PressPermis{100}:=[FALSE,FALSE,FALSE,FALSE,FALSE,FALSE,FALSE,FALSE,FALSE,FALSE,FALSE,FALSE,FALSE,FALSE,FALSE,FALSE,FALSE,FALSE,FALSE,FALSE,FALSE,FALSE,FALSE,FALSE,FALSE,FALSE,FALSE,FALSE,FALSE,FALSE,FALSE,FALSE,FALSE,FALSE,FALSE,FALSE,FALSE,FALSE,FALSE,FALSE,FALSE,FALSE,FALSE,FALSE,FALSE,FALSE,FALSE,FALSE,FALSE,FALSE,FALSE,FALSE,FALSE,FALSE,FALSE,FALSE,FALSE,FALSE,FALSE,FALSE,FALSE,FALSE,FALSE,FALSE,FALSE,FALSE,FALSE,FALSE,FALSE,FALSE,FALSE,FALSE,FALSE,FALSE,FALSE,FALSE,FALSE,FALSE,FALSE,FALSE,FALSE,FALSE,FALSE,FALSE,FALSE,FALSE,FALSE,FALSE,FALSE,FALSE,FALSE,FALSE,FALSE,FALSE,FALSE,FALSE,FALSE,FALSE,FALSE,FALSE];
    PERS num PutOffestNum{100}:=[0,0,0,0,0,0,0,0,0,0,0,0,0,0,0,0,0,0,0,0,0,0,0,0,0,0,0,0,0,0,0,0,0,0,0,0,0,0,0,0,0,0,0,0,0,0,0,0,0,0,0,0,0,0,0,0,0,0,0,0,0,0,0,0,0,0,0,0,0,0,0,0,0,0,0,0,0,0,0,0,0,0,0,0,0,0,0,0,0,0,0,0,0,0,0,0,0,0,0,0];
    !==============================================================================

    !======================OffsetData==============================================
    PERS num FCDisBigN:=1;
    PERS num FCDisSmallN:=1;
    PERS num FCyDisBigN:=1;
    PERS num FCyDisSmallN:=1;
    PERS bool FCDisBig:=FALSE;
    PERS bool FCDisSmall:=FALSE;
    PERS num offestNum:=0;
    PERS num offestNumT:=10;
    PERS num offestNumData:=0.2;
    !==============================================================================

    !=====================ForceData================================================
    PERS num Force_out_x:=90;
    PERS num Force_out_y:=179.597;
    PERS num Force_out_z:=431.599;
    !==============================================================================

    !====================MainRoutData==============================================
    PERS num TestNum;
    PERS num MaxTestTimes:=10;
    PERS num ActionTimes:=0;
    PERS num DataIndex:=1;
    PERS bool FirstPress:=TRUE;
    PERS robtarget FirstPoint;
    PERS num MOffsetNum;
    PERS num i:=3;
    PERS string ad:="asas";
    PERS string MoveType{100}:=["","","","","","","","","","","","","","","","","","","","","","","","","","","","","","","","","","","","","","","","","","","","","","","","","","","","","","","","","","","","","","","","","","","","","","","","","","","","","","","","","","","","","","","","","","","","","","","","","","","",""];
    PERS robtarget PointC{100}:=[[[943.59,288.91,1103.35],[0.5,9.08645E-7,0.866025,-1.01075E-6],[0,-1,0,0],[9E+9,9E+9,9E+9,9E+9,9E+9,9E+9]],[[943.59,288.91,1103.35],[0.5,9.08645E-7,0.866025,-1.01075E-6],[0,-1,0,0],[9E+9,9E+9,9E+9,9E+9,9E+9,9E+9]],[[943.59,288.91,1103.35],[0.5,9.08645E-7,0.866025,-1.01075E-6],[0,-1,0,0],[9E+9,9E+9,9E+9,9E+9,9E+9,9E+9]],[[943.59,288.91,1103.35],[0.5,9.08645E-7,0.866025,-1.01075E-6],[0,-1,0,0],[9E+9,9E+9,9E+9,9E+9,9E+9,9E+9]],[[943.59,288.91,1103.35],[0.5,9.08645E-7,0.866025,-1.01075E-6],[0,-1,0,0],[9E+9,9E+9,9E+9,9E+9,9E+9,9E+9]],[[943.59,288.91,1103.35],[0.5,9.08645E-7,0.866025,-1.01075E-6],[0,-1,0,0],[9E+9,9E+9,9E+9,9E+9,9E+9,9E+9]],[[943.59,288.91,1103.35],[0.5,9.08645E-7,0.866025,-1.01075E-6],[0,-1,0,0],[9E+9,9E+9,9E+9,9E+9,9E+9,9E+9]],[[943.59,288.91,1103.35],[0.5,9.08645E-7,0.866025,-1.01075E-6],[0,-1,0,0],[9E+9,9E+9,9E+9,9E+9,9E+9,9E+9]],[[943.59,288.91,1103.35],[0.5,9.08645E-7,0.866025,-1.01075E-6],[0,-1,0,0],[9E+9,9E+9,9E+9,9E+9,9E+9,9E+9]],[[943.59,288.91,1103.35],[0.5,9.08645E-7,0.866025,-1.01075E-6],[0,-1,0,0],[9E+9,9E+9,9E+9,9E+9,9E+9,9E+9]],[[943.59,288.91,1103.35],[0.5,9.08645E-7,0.866025,-1.01075E-6],[0,-1,0,0],[9E+9,9E+9,9E+9,9E+9,9E+9,9E+9]],[[943.59,288.91,1103.35],[0.5,9.08645E-7,0.866025,-1.01075E-6],[0,-1,0,0],[9E+9,9E+9,9E+9,9E+9,9E+9,9E+9]],[[943.59,288.91,1103.35],[0.5,9.08645E-7,0.866025,-1.01075E-6],[0,-1,0,0],[9E+9,9E+9,9E+9,9E+9,9E+9,9E+9]],[[943.59,288.91,1103.35],[0.5,9.08645E-7,0.866025,-1.01075E-6],[0,-1,0,0],[9E+9,9E+9,9E+9,9E+9,9E+9,9E+9]],[[943.59,288.91,1103.35],[0.5,9.08645E-7,0.866025,-1.01075E-6],[0,-1,0,0],[9E+9,9E+9,9E+9,9E+9,9E+9,9E+9]],[[943.59,288.91,1103.35],[0.5,9.08645E-7,0.866025,-1.01075E-6],[0,-1,0,0],[9E+9,9E+9,9E+9,9E+9,9E+9,9E+9]],[[943.59,288.91,1103.35],[0.5,9.08645E-7,0.866025,-1.01075E-6],[0,-1,0,0],[9E+9,9E+9,9E+9,9E+9,9E+9,9E+9]],[[943.59,288.91,1103.35],[0.5,9.08645E-7,0.866025,-1.01075E-6],[0,-1,0,0],[9E+9,9E+9,9E+9,9E+9,9E+9,9E+9]],[[943.59,288.91,1103.35],[0.5,9.08645E-7,0.866025,-1.01075E-6],[0,-1,0,0],[9E+9,9E+9,9E+9,9E+9,9E+9,9E+9]],[[943.59,288.91,1103.35],[0.5,9.08645E-7,0.866025,-1.01075E-6],[0,-1,0,0],[9E+9,9E+9,9E+9,9E+9,9E+9,9E+9]],[[943.59,288.91,1103.35],[0.5,9.08645E-7,0.866025,-1.01075E-6],[0,-1,0,0],[9E+9,9E+9,9E+9,9E+9,9E+9,9E+9]],[[943.59,288.91,1103.35],[0.5,9.08645E-7,0.866025,-1.01075E-6],[0,-1,0,0],[9E+9,9E+9,9E+9,9E+9,9E+9,9E+9]],[[943.59,288.91,1103.35],[0.5,9.08645E-7,0.866025,-1.01075E-6],[0,-1,0,0],[9E+9,9E+9,9E+9,9E+9,9E+9,9E+9]],[[943.59,288.91,1103.35],[0.5,9.08645E-7,0.866025,-1.01075E-6],[0,-1,0,0],[9E+9,9E+9,9E+9,9E+9,9E+9,9E+9]],[[943.59,288.91,1103.35],[0.5,9.08645E-7,0.866025,-1.01075E-6],[0,-1,0,0],[9E+9,9E+9,9E+9,9E+9,9E+9,9E+9]],[[943.59,288.91,1103.35],[0.5,9.08645E-7,0.866025,-1.01075E-6],[0,-1,0,0],[9E+9,9E+9,9E+9,9E+9,9E+9,9E+9]],[[943.59,288.91,1103.35],[0.5,9.08645E-7,0.866025,-1.01075E-6],[0,-1,0,0],[9E+9,9E+9,9E+9,9E+9,9E+9,9E+9]],[[943.59,288.91,1103.35],[0.5,9.08645E-7,0.866025,-1.01075E-6],[0,-1,0,0],[9E+9,9E+9,9E+9,9E+9,9E+9,9E+9]],[[943.59,288.91,1103.35],[0.5,9.08645E-7,0.866025,-1.01075E-6],[0,-1,0,0],[9E+9,9E+9,9E+9,9E+9,9E+9,9E+9]],[[943.59,288.91,1103.35],[0.5,9.08645E-7,0.866025,-1.01075E-6],[0,-1,0,0],[9E+9,9E+9,9E+9,9E+9,9E+9,9E+9]],[[943.59,288.91,1103.35],[0.5,9.08645E-7,0.866025,-1.01075E-6],[0,-1,0,0],[9E+9,9E+9,9E+9,9E+9,9E+9,9E+9]],[[943.59,288.91,1103.35],[0.5,9.08645E-7,0.866025,-1.01075E-6],[0,-1,0,0],[9E+9,9E+9,9E+9,9E+9,9E+9,9E+9]],[[943.59,288.91,1103.35],[0.5,9.08645E-7,0.866025,-1.01075E-6],[0,-1,0,0],[9E+9,9E+9,9E+9,9E+9,9E+9,9E+9]],[[943.59,288.91,1103.35],[0.5,9.08645E-7,0.866025,-1.01075E-6],[0,-1,0,0],[9E+9,9E+9,9E+9,9E+9,9E+9,9E+9]],[[943.59,288.91,1103.35],[0.5,9.08645E-7,0.866025,-1.01075E-6],[0,-1,0,0],[9E+9,9E+9,9E+9,9E+9,9E+9,9E+9]],[[943.59,288.91,1103.35],[0.5,9.08645E-7,0.866025,-1.01075E-6],[0,-1,0,0],[9E+9,9E+9,9E+9,9E+9,9E+9,9E+9]],[[943.59,288.91,1103.35],[0.5,9.08645E-7,0.866025,-1.01075E-6],[0,-1,0,0],[9E+9,9E+9,9E+9,9E+9,9E+9,9E+9]],[[943.59,288.91,1103.35],[0.5,9.08645E-7,0.866025,-1.01075E-6],[0,-1,0,0],[9E+9,9E+9,9E+9,9E+9,9E+9,9E+9]],[[943.59,288.91,1103.35],[0.5,9.08645E-7,0.866025,-1.01075E-6],[0,-1,0,0],[9E+9,9E+9,9E+9,9E+9,9E+9,9E+9]],[[943.59,288.91,1103.35],[0.5,9.08645E-7,0.866025,-1.01075E-6],[0,-1,0,0],[9E+9,9E+9,9E+9,9E+9,9E+9,9E+9]],[[943.59,288.91,1103.35],[0.5,9.08645E-7,0.866025,-1.01075E-6],[0,-1,0,0],[9E+9,9E+9,9E+9,9E+9,9E+9,9E+9]],[[943.59,288.91,1103.35],[0.5,9.08645E-7,0.866025,-1.01075E-6],[0,-1,0,0],[9E+9,9E+9,9E+9,9E+9,9E+9,9E+9]],[[943.59,288.91,1103.35],[0.5,9.08645E-7,0.866025,-1.01075E-6],[0,-1,0,0],[9E+9,9E+9,9E+9,9E+9,9E+9,9E+9]],[[943.59,288.91,1103.35],[0.5,9.08645E-7,0.866025,-1.01075E-6],[0,-1,0,0],[9E+9,9E+9,9E+9,9E+9,9E+9,9E+9]],[[943.59,288.91,1103.35],[0.5,9.08645E-7,0.866025,-1.01075E-6],[0,-1,0,0],[9E+9,9E+9,9E+9,9E+9,9E+9,9E+9]],[[943.59,288.91,1103.35],[0.5,9.08645E-7,0.866025,-1.01075E-6],[0,-1,0,0],[9E+9,9E+9,9E+9,9E+9,9E+9,9E+9]],[[943.59,288.91,1103.35],[0.5,9.08645E-7,0.866025,-1.01075E-6],[0,-1,0,0],[9E+9,9E+9,9E+9,9E+9,9E+9,9E+9]],[[943.59,288.91,1103.35],[0.5,9.08645E-7,0.866025,-1.01075E-6],[0,-1,0,0],[9E+9,9E+9,9E+9,9E+9,9E+9,9E+9]],[[943.59,288.91,1103.35],[0.5,9.08645E-7,0.866025,-1.01075E-6],[0,-1,0,0],[9E+9,9E+9,9E+9,9E+9,9E+9,9E+9]],[[943.59,288.91,1103.35],[0.5,9.08645E-7,0.866025,-1.01075E-6],[0,-1,0,0],[9E+9,9E+9,9E+9,9E+9,9E+9,9E+9]],[[943.59,288.91,1103.35],[0.5,9.08645E-7,0.866025,-1.01075E-6],[0,-1,0,0],[9E+9,9E+9,9E+9,9E+9,9E+9,9E+9]],[[943.59,288.91,1103.35],[0.5,9.08645E-7,0.866025,-1.01075E-6],[0,-1,0,0],[9E+9,9E+9,9E+9,9E+9,9E+9,9E+9]],[[943.59,288.91,1103.35],[0.5,9.08645E-7,0.866025,-1.01075E-6],[0,-1,0,0],[9E+9,9E+9,9E+9,9E+9,9E+9,9E+9]],[[943.59,288.91,1103.35],[0.5,9.08645E-7,0.866025,-1.01075E-6],[0,-1,0,0],[9E+9,9E+9,9E+9,9E+9,9E+9,9E+9]],[[943.59,288.91,1103.35],[0.5,9.08645E-7,0.866025,-1.01075E-6],[0,-1,0,0],[9E+9,9E+9,9E+9,9E+9,9E+9,9E+9]],[[943.59,288.91,1103.35],[0.5,9.08645E-7,0.866025,-1.01075E-6],[0,-1,0,0],[9E+9,9E+9,9E+9,9E+9,9E+9,9E+9]],[[943.59,288.91,1103.35],[0.5,9.08645E-7,0.866025,-1.01075E-6],[0,-1,0,0],[9E+9,9E+9,9E+9,9E+9,9E+9,9E+9]],[[943.59,288.91,1103.35],[0.5,9.08645E-7,0.866025,-1.01075E-6],[0,-1,0,0],[9E+9,9E+9,9E+9,9E+9,9E+9,9E+9]],[[943.59,288.91,1103.35],[0.5,9.08645E-7,0.866025,-1.01075E-6],[0,-1,0,0],[9E+9,9E+9,9E+9,9E+9,9E+9,9E+9]],[[943.59,288.91,1103.35],[0.5,9.08645E-7,0.866025,-1.01075E-6],[0,-1,0,0],[9E+9,9E+9,9E+9,9E+9,9E+9,9E+9]],[[943.59,288.91,1103.35],[0.5,9.08645E-7,0.866025,-1.01075E-6],[0,-1,0,0],[9E+9,9E+9,9E+9,9E+9,9E+9,9E+9]],[[943.59,288.91,1103.35],[0.5,9.08645E-7,0.866025,-1.01075E-6],[0,-1,0,0],[9E+9,9E+9,9E+9,9E+9,9E+9,9E+9]],[[943.59,288.91,1103.35],[0.5,9.08645E-7,0.866025,-1.01075E-6],[0,-1,0,0],[9E+9,9E+9,9E+9,9E+9,9E+9,9E+9]],[[943.59,288.91,1103.35],[0.5,9.08645E-7,0.866025,-1.01075E-6],[0,-1,0,0],[9E+9,9E+9,9E+9,9E+9,9E+9,9E+9]],[[943.59,288.91,1103.35],[0.5,9.08645E-7,0.866025,-1.01075E-6],[0,-1,0,0],[9E+9,9E+9,9E+9,9E+9,9E+9,9E+9]],[[943.59,288.91,1103.35],[0.5,9.08645E-7,0.866025,-1.01075E-6],[0,-1,0,0],[9E+9,9E+9,9E+9,9E+9,9E+9,9E+9]],[[943.59,288.91,1103.35],[0.5,9.08645E-7,0.866025,-1.01075E-6],[0,-1,0,0],[9E+9,9E+9,9E+9,9E+9,9E+9,9E+9]],[[943.59,288.91,1103.35],[0.5,9.08645E-7,0.866025,-1.01075E-6],[0,-1,0,0],[9E+9,9E+9,9E+9,9E+9,9E+9,9E+9]],[[943.59,288.91,1103.35],[0.5,9.08645E-7,0.866025,-1.01075E-6],[0,-1,0,0],[9E+9,9E+9,9E+9,9E+9,9E+9,9E+9]],[[943.59,288.91,1103.35],[0.5,9.08645E-7,0.866025,-1.01075E-6],[0,-1,0,0],[9E+9,9E+9,9E+9,9E+9,9E+9,9E+9]],[[943.59,288.91,1103.35],[0.5,9.08645E-7,0.866025,-1.01075E-6],[0,-1,0,0],[9E+9,9E+9,9E+9,9E+9,9E+9,9E+9]],[[943.59,288.91,1103.35],[0.5,9.08645E-7,0.866025,-1.01075E-6],[0,-1,0,0],[9E+9,9E+9,9E+9,9E+9,9E+9,9E+9]],[[943.59,288.91,1103.35],[0.5,9.08645E-7,0.866025,-1.01075E-6],[0,-1,0,0],[9E+9,9E+9,9E+9,9E+9,9E+9,9E+9]],[[943.59,288.91,1103.35],[0.5,9.08645E-7,0.866025,-1.01075E-6],[0,-1,0,0],[9E+9,9E+9,9E+9,9E+9,9E+9,9E+9]],[[943.59,288.91,1103.35],[0.5,9.08645E-7,0.866025,-1.01075E-6],[0,-1,0,0],[9E+9,9E+9,9E+9,9E+9,9E+9,9E+9]],[[943.59,288.91,1103.35],[0.5,9.08645E-7,0.866025,-1.01075E-6],[0,-1,0,0],[9E+9,9E+9,9E+9,9E+9,9E+9,9E+9]],[[943.59,288.91,1103.35],[0.5,9.08645E-7,0.866025,-1.01075E-6],[0,-1,0,0],[9E+9,9E+9,9E+9,9E+9,9E+9,9E+9]],[[943.59,288.91,1103.35],[0.5,9.08645E-7,0.866025,-1.01075E-6],[0,-1,0,0],[9E+9,9E+9,9E+9,9E+9,9E+9,9E+9]],[[943.59,288.91,1103.35],[0.5,9.08645E-7,0.866025,-1.01075E-6],[0,-1,0,0],[9E+9,9E+9,9E+9,9E+9,9E+9,9E+9]],[[943.59,288.91,1103.35],[0.5,9.08645E-7,0.866025,-1.01075E-6],[0,-1,0,0],[9E+9,9E+9,9E+9,9E+9,9E+9,9E+9]],[[943.59,288.91,1103.35],[0.5,9.08645E-7,0.866025,-1.01075E-6],[0,-1,0,0],[9E+9,9E+9,9E+9,9E+9,9E+9,9E+9]],[[943.59,288.91,1103.35],[0.5,9.08645E-7,0.866025,-1.01075E-6],[0,-1,0,0],[9E+9,9E+9,9E+9,9E+9,9E+9,9E+9]],[[943.59,288.91,1103.35],[0.5,9.08645E-7,0.866025,-1.01075E-6],[0,-1,0,0],[9E+9,9E+9,9E+9,9E+9,9E+9,9E+9]],[[943.59,288.91,1103.35],[0.5,9.08645E-7,0.866025,-1.01075E-6],[0,-1,0,0],[9E+9,9E+9,9E+9,9E+9,9E+9,9E+9]],[[943.59,288.91,1103.35],[0.5,9.08645E-7,0.866025,-1.01075E-6],[0,-1,0,0],[9E+9,9E+9,9E+9,9E+9,9E+9,9E+9]],[[943.59,288.91,1103.35],[0.5,9.08645E-7,0.866025,-1.01075E-6],[0,-1,0,0],[9E+9,9E+9,9E+9,9E+9,9E+9,9E+9]],[[943.59,288.91,1103.35],[0.5,9.08645E-7,0.866025,-1.01075E-6],[0,-1,0,0],[9E+9,9E+9,9E+9,9E+9,9E+9,9E+9]],[[943.59,288.91,1103.35],[0.5,9.08645E-7,0.866025,-1.01075E-6],[0,-1,0,0],[9E+9,9E+9,9E+9,9E+9,9E+9,9E+9]],[[943.59,288.91,1103.35],[0.5,9.08645E-7,0.866025,-1.01075E-6],[0,-1,0,0],[9E+9,9E+9,9E+9,9E+9,9E+9,9E+9]],[[943.59,288.91,1103.35],[0.5,9.08645E-7,0.866025,-1.01075E-6],[0,-1,0,0],[9E+9,9E+9,9E+9,9E+9,9E+9,9E+9]],[[943.59,288.91,1103.35],[0.5,9.08645E-7,0.866025,-1.01075E-6],[0,-1,0,0],[9E+9,9E+9,9E+9,9E+9,9E+9,9E+9]],[[943.59,288.91,1103.35],[0.5,9.08645E-7,0.866025,-1.01075E-6],[0,-1,0,0],[9E+9,9E+9,9E+9,9E+9,9E+9,9E+9]],[[943.59,288.91,1103.35],[0.5,9.08645E-7,0.866025,-1.01075E-6],[0,-1,0,0],[9E+9,9E+9,9E+9,9E+9,9E+9,9E+9]],[[943.59,288.91,1103.35],[0.5,9.08645E-7,0.866025,-1.01075E-6],[0,-1,0,0],[9E+9,9E+9,9E+9,9E+9,9E+9,9E+9]],[[943.59,288.91,1103.35],[0.5,9.08645E-7,0.866025,-1.01075E-6],[0,-1,0,0],[9E+9,9E+9,9E+9,9E+9,9E+9,9E+9]],[[943.59,288.91,1103.35],[0.5,9.08645E-7,0.866025,-1.01075E-6],[0,-1,0,0],[9E+9,9E+9,9E+9,9E+9,9E+9,9E+9]],[[943.59,288.91,1103.35],[0.5,9.08645E-7,0.866025,-1.01075E-6],[0,-1,0,0],[9E+9,9E+9,9E+9,9E+9,9E+9,9E+9]],[[943.59,288.91,1103.35],[0.5,9.08645E-7,0.866025,-1.01075E-6],[0,-1,0,0],[9E+9,9E+9,9E+9,9E+9,9E+9,9E+9]],[[943.59,288.91,1103.35],[0.5,9.08645E-7,0.866025,-1.01075E-6],[0,-1,0,0],[9E+9,9E+9,9E+9,9E+9,9E+9,9E+9]],[[943.59,288.91,1103.35],[0.5,9.08645E-7,0.866025,-1.01075E-6],[0,-1,0,0],[9E+9,9E+9,9E+9,9E+9,9E+9,9E+9]]];
    PERS bool JudgeWaitStartSign{100,3}:=[[FALSE,FALSE,FALSE],[FALSE,FALSE,FALSE],[FALSE,FALSE,FALSE],[FALSE,FALSE,FALSE],[FALSE,FALSE,FALSE],[FALSE,FALSE,FALSE],[FALSE,FALSE,FALSE],[FALSE,FALSE,FALSE],[FALSE,FALSE,FALSE],[TRUE,FALSE,FALSE],[FALSE,FALSE,FALSE],[FALSE,FALSE,FALSE],[FALSE,FALSE,FALSE],[FALSE,FALSE,FALSE],[FALSE,FALSE,FALSE],[FALSE,FALSE,FALSE],[FALSE,FALSE,FALSE],[FALSE,FALSE,FALSE],[FALSE,FALSE,FALSE],[FALSE,FALSE,FALSE],[FALSE,FALSE,FALSE],[FALSE,FALSE,FALSE],[FALSE,FALSE,FALSE],[FALSE,FALSE,FALSE],[FALSE,FALSE,FALSE],[FALSE,FALSE,FALSE],[FALSE,FALSE,FALSE],[FALSE,FALSE,FALSE],[FALSE,FALSE,FALSE],[FALSE,FALSE,FALSE],[FALSE,FALSE,FALSE],[FALSE,FALSE,FALSE],[FALSE,FALSE,FALSE],[FALSE,FALSE,FALSE],[FALSE,FALSE,FALSE],[FALSE,FALSE,FALSE],[FALSE,FALSE,FALSE],[FALSE,FALSE,FALSE],[FALSE,FALSE,FALSE],[FALSE,FALSE,FALSE],[FALSE,FALSE,FALSE],[FALSE,FALSE,FALSE],[FALSE,FALSE,FALSE],[FALSE,FALSE,FALSE],[FALSE,FALSE,FALSE],[FALSE,FALSE,FALSE],[FALSE,FALSE,FALSE],[FALSE,FALSE,FALSE],[FALSE,FALSE,FALSE],[FALSE,FALSE,FALSE],[FALSE,FALSE,FALSE],[FALSE,FALSE,FALSE],[FALSE,FALSE,FALSE],[FALSE,FALSE,FALSE],[FALSE,FALSE,FALSE],[FALSE,FALSE,FALSE],[FALSE,FALSE,FALSE],[FALSE,FALSE,FALSE],[FALSE,FALSE,FALSE],[FALSE,FALSE,FALSE],[FALSE,FALSE,FALSE],[FALSE,FALSE,FALSE],[FALSE,FALSE,FALSE],[FALSE,FALSE,FALSE],[FALSE,FALSE,FALSE],[FALSE,FALSE,FALSE],[FALSE,FALSE,FALSE],[FALSE,FALSE,FALSE],[FALSE,FALSE,FALSE],[FALSE,FALSE,FALSE],[FALSE,FALSE,FALSE],[FALSE,FALSE,FALSE],[FALSE,FALSE,FALSE],[FALSE,FALSE,FALSE],[FALSE,FALSE,FALSE],[FALSE,FALSE,FALSE],[FALSE,FALSE,FALSE],[FALSE,FALSE,FALSE],[FALSE,FALSE,FALSE],[FALSE,FALSE,FALSE],[FALSE,FALSE,FALSE],[FALSE,FALSE,FALSE],[FALSE,FALSE,FALSE],[FALSE,FALSE,FALSE],[FALSE,FALSE,FALSE],[FALSE,FALSE,FALSE],[FALSE,FALSE,FALSE],[FALSE,FALSE,FALSE],[FALSE,FALSE,FALSE],[FALSE,FALSE,FALSE],[FALSE,FALSE,FALSE],[FALSE,FALSE,FALSE],[FALSE,FALSE,FALSE],[FALSE,FALSE,FALSE],[FALSE,FALSE,FALSE],[FALSE,FALSE,FALSE],[FALSE,FALSE,FALSE],[FALSE,FALSE,FALSE],[FALSE,FALSE,FALSE],[FALSE,FALSE,FALSE]];
    PERS bool JudgeWaitMidSign{100,3}:=[[FALSE,FALSE,FALSE],[TRUE,FALSE,FALSE],[FALSE,FALSE,FALSE],[FALSE,FALSE,FALSE],[FALSE,FALSE,FALSE],[FALSE,FALSE,FALSE],[FALSE,FALSE,FALSE],[FALSE,FALSE,FALSE],[FALSE,FALSE,FALSE],[TRUE,FALSE,FALSE],[FALSE,FALSE,FALSE],[FALSE,FALSE,FALSE],[FALSE,FALSE,FALSE],[FALSE,FALSE,FALSE],[FALSE,FALSE,FALSE],[FALSE,FALSE,FALSE],[FALSE,FALSE,FALSE],[FALSE,FALSE,FALSE],[FALSE,FALSE,FALSE],[FALSE,FALSE,FALSE],[FALSE,FALSE,FALSE],[FALSE,FALSE,FALSE],[FALSE,FALSE,FALSE],[FALSE,FALSE,FALSE],[FALSE,FALSE,FALSE],[FALSE,FALSE,FALSE],[FALSE,FALSE,FALSE],[FALSE,FALSE,FALSE],[FALSE,FALSE,FALSE],[FALSE,FALSE,FALSE],[FALSE,FALSE,FALSE],[FALSE,FALSE,FALSE],[FALSE,FALSE,FALSE],[FALSE,FALSE,FALSE],[FALSE,FALSE,FALSE],[FALSE,FALSE,FALSE],[FALSE,FALSE,FALSE],[FALSE,FALSE,FALSE],[FALSE,FALSE,FALSE],[FALSE,FALSE,FALSE],[FALSE,FALSE,FALSE],[FALSE,FALSE,FALSE],[FALSE,FALSE,FALSE],[FALSE,FALSE,FALSE],[FALSE,FALSE,FALSE],[FALSE,FALSE,FALSE],[FALSE,FALSE,FALSE],[FALSE,FALSE,FALSE],[FALSE,FALSE,FALSE],[FALSE,FALSE,FALSE],[FALSE,FALSE,FALSE],[FALSE,FALSE,FALSE],[FALSE,FALSE,FALSE],[FALSE,FALSE,FALSE],[FALSE,FALSE,FALSE],[FALSE,FALSE,FALSE],[FALSE,FALSE,FALSE],[FALSE,FALSE,FALSE],[FALSE,FALSE,FALSE],[FALSE,FALSE,FALSE],[FALSE,FALSE,FALSE],[FALSE,FALSE,FALSE],[FALSE,FALSE,FALSE],[FALSE,FALSE,FALSE],[FALSE,FALSE,FALSE],[FALSE,FALSE,FALSE],[FALSE,FALSE,FALSE],[FALSE,FALSE,FALSE],[FALSE,FALSE,FALSE],[FALSE,FALSE,FALSE],[FALSE,FALSE,FALSE],[FALSE,FALSE,FALSE],[FALSE,FALSE,FALSE],[FALSE,FALSE,FALSE],[FALSE,FALSE,FALSE],[FALSE,FALSE,FALSE],[FALSE,FALSE,FALSE],[FALSE,FALSE,FALSE],[FALSE,FALSE,FALSE],[FALSE,FALSE,FALSE],[FALSE,FALSE,FALSE],[FALSE,FALSE,FALSE],[FALSE,FALSE,FALSE],[FALSE,FALSE,FALSE],[FALSE,FALSE,FALSE],[FALSE,FALSE,FALSE],[FALSE,FALSE,FALSE],[FALSE,FALSE,FALSE],[FALSE,FALSE,FALSE],[FALSE,FALSE,FALSE],[FALSE,FALSE,FALSE],[FALSE,FALSE,FALSE],[FALSE,FALSE,FALSE],[FALSE,FALSE,FALSE],[FALSE,FALSE,FALSE],[FALSE,FALSE,FALSE],[FALSE,FALSE,FALSE],[FALSE,FALSE,FALSE],[FALSE,FALSE,FALSE],[FALSE,FALSE,FALSE]];
    PERS string JudgeWaitSignal{100}:=["23","","","","","","","","","","","","","","","","","","","","","","","","","","","","","","","","","","","","","","","","","","","","","","","","","","","","","","","","","","","","","","","","","","","","","","","","","","","","","","","","","","","","","","","","","","","","","","","","","","",""];
    PERS bool SelectActionReset{100,3}:=[[FALSE,FALSE,FALSE],[FALSE,FALSE,FALSE],[FALSE,FALSE,FALSE],[FALSE,FALSE,FALSE],[FALSE,FALSE,FALSE],[FALSE,FALSE,FALSE],[FALSE,FALSE,FALSE],[FALSE,FALSE,FALSE],[FALSE,FALSE,FALSE],[FALSE,FALSE,FALSE],[FALSE,FALSE,FALSE],[FALSE,FALSE,FALSE],[FALSE,FALSE,FALSE],[FALSE,FALSE,FALSE],[FALSE,FALSE,FALSE],[FALSE,FALSE,FALSE],[FALSE,FALSE,FALSE],[FALSE,FALSE,FALSE],[FALSE,FALSE,FALSE],[FALSE,FALSE,FALSE],[FALSE,FALSE,FALSE],[FALSE,FALSE,FALSE],[FALSE,FALSE,FALSE],[FALSE,FALSE,FALSE],[FALSE,FALSE,FALSE],[FALSE,FALSE,FALSE],[FALSE,FALSE,FALSE],[FALSE,FALSE,FALSE],[FALSE,FALSE,FALSE],[FALSE,FALSE,FALSE],[FALSE,FALSE,FALSE],[FALSE,FALSE,FALSE],[FALSE,FALSE,FALSE],[FALSE,FALSE,FALSE],[FALSE,FALSE,FALSE],[FALSE,FALSE,FALSE],[FALSE,FALSE,FALSE],[FALSE,FALSE,FALSE],[FALSE,FALSE,FALSE],[FALSE,FALSE,FALSE],[FALSE,FALSE,FALSE],[FALSE,FALSE,FALSE],[FALSE,FALSE,FALSE],[FALSE,FALSE,FALSE],[FALSE,FALSE,FALSE],[FALSE,FALSE,FALSE],[FALSE,FALSE,FALSE],[FALSE,FALSE,FALSE],[FALSE,FALSE,FALSE],[FALSE,FALSE,FALSE],[FALSE,FALSE,FALSE],[FALSE,FALSE,FALSE],[FALSE,FALSE,FALSE],[FALSE,FALSE,FALSE],[FALSE,FALSE,FALSE],[FALSE,FALSE,FALSE],[FALSE,FALSE,FALSE],[FALSE,FALSE,FALSE],[FALSE,FALSE,FALSE],[FALSE,FALSE,FALSE],[FALSE,FALSE,FALSE],[FALSE,FALSE,FALSE],[FALSE,FALSE,FALSE],[FALSE,FALSE,FALSE],[FALSE,FALSE,FALSE],[FALSE,FALSE,FALSE],[FALSE,FALSE,FALSE],[FALSE,FALSE,FALSE],[FALSE,FALSE,FALSE],[FALSE,FALSE,FALSE],[FALSE,FALSE,FALSE],[FALSE,FALSE,FALSE],[FALSE,FALSE,FALSE],[FALSE,FALSE,FALSE],[FALSE,FALSE,FALSE],[FALSE,FALSE,FALSE],[FALSE,FALSE,FALSE],[FALSE,FALSE,FALSE],[FALSE,FALSE,FALSE],[FALSE,FALSE,FALSE],[FALSE,FALSE,FALSE],[FALSE,FALSE,FALSE],[FALSE,FALSE,FALSE],[FALSE,FALSE,FALSE],[FALSE,FALSE,FALSE],[FALSE,FALSE,FALSE],[FALSE,FALSE,FALSE],[FALSE,FALSE,FALSE],[FALSE,FALSE,FALSE],[FALSE,FALSE,FALSE],[FALSE,FALSE,FALSE],[FALSE,FALSE,FALSE],[FALSE,FALSE,FALSE],[FALSE,FALSE,FALSE],[FALSE,FALSE,FALSE],[FALSE,FALSE,FALSE],[FALSE,FALSE,FALSE],[FALSE,FALSE,FALSE],[FALSE,FALSE,FALSE],[FALSE,FALSE,FALSE]];
    !==============================================================================
ENDMODULE

--- Backups/DeskSystem/SYSPAR/EIO.cfg ---
EIO:CFG_1.0:6:1::
#
INDUSTRIAL_NETWORK:

      -Name "PROFINET" -Connection "PROFINET Network"\
      -Label "PROFINET Controller/Device Network" -StationName ""
#
PROFINET_DRIVER:

      -Name "PROFINET_COMMON_DATA"
#
PROFINET_INTERNAL_DEVICE:

      -Name "PN_Internal_Device" -VendorName "ABB Robotics"\
      -ProductName "PROFINET Internal Device"
#
EIO_SIGNAL:

      -Name "DO_FCylinder" -SignalType "DO" -Device "PN_Internal_Device"\
      -DeviceMap "0" -Access "All"

      -Name "DO_SCylinder" -SignalType "DO" -Device "PN_Internal_Device"\
      -DeviceMap "1" -Access "All"

      -Name "DO_TCylinder" -SignalType "DO" -Device "PN_Internal_Device"\
      -DeviceMap "2" -Access "All"

      -Name "OffestAlarmOn" -SignalType "DO" -Access "All"

      -Name "DI_FCylinder" -SignalType "DI" -Device "PN_Internal_Device"\
      -DeviceMap "0" -Access "All"

      -Name "DI_SCylinder" -SignalType "DI" -Device "PN_Internal_Device"\
      -DeviceMap "1" -Access "All"

      -Name "DI_TCylinder" -SignalType "DI" -Device "PN_Internal_Device"\
      -DeviceMap "2" -Access "All"

      -Name "DO_SignReset" -SignalType "DO" -Access "All"

      -Name "DI_CarReady" -SignalType "DI"

      -Name "DI_PLCOK" -SignalType "DI"

      -Name "DI_CarWindowOpen" -SignalType "DI"

      -Name "DI_FMCylinder" -SignalType "DI" -Device "PN_Internal_Device"\
      -DeviceMap "3" -Access "All"

      -Name "DI_SMCylinder" -SignalType "DI" -Device "PN_Internal_Device"\
      -DeviceMap "4" -Access "All"

      -Name "DI_TMCylinder" -SignalType "DI" -Device "PN_Internal_Device"\
      -DeviceMap "5" -Access "All"
